// TIA Portal V16 export
// export: Created 2022-11-17T15:49:43.8022431Z, ExportSetting WithDefaults, DisplayName Totally Integrated Automation Portal, DisplayVersion V16 Update 6, DisplayName TIA Portal Version Control Interface, DisplayVersion V16 Update 2, DisplayName TIA Portal Openness, DisplayVersion V16 Update 6, DisplayName SINAMICS Startdrive Advanced, DisplayVersion V16 Update 5, DisplayName SINAMICS Startdrive G130, G150, S120, S150, SINAMICS MV, S210, DisplayVersion V16 Update 5, DisplayName SINAMICS Startdrive G110M, G120, G120C, G120D, G120P, G115D, DisplayVersion V16 Update 5, DisplayName STEP 7 Professional, DisplayVersion V16 Update 6, DisplayName STEP 7 Safety, DisplayVersion V16, DisplayName WinCC Advanced, DisplayVersion V16 Update 6
DATA_BLOCK "DB237_Program13"   // DB237
{ S7_Optimized_Access := 'FALSE' }
AUTHOR : Robopac
VERSION : 0.0
// stored: AutoNumber false, IsOnlyStoredInLoadMemory false, IsWriteProtectedInAS false
   VAR RETAIN
      Program13 { S7_SetPoint := 'True'} : "DatiProgramma";
   END_VAR
BEGIN
   Program13.Wrapping := TRUE;
   Program13.TopLenght := 500;
   Program13.TopRelease := 0;
   Program13.TopDown := 0;
   Program13.Top := 4;
   Program13.PressurePTime := 0;
   Program13.LifterTime := 0;
   Program13.RevOverContrast := 1;
   Program13.RopeEndCycle := 16#02;
   Program13.Spare4 := 16#01;
   Program13.RopeTime := 1500;
   Program13.RevOverClamp := 1;
   Program13.FilmForceFinalRev := 10;
   Program13.FilmPrestretchFinalRev := 100;
   Program13.ArmSpeed := 100;
   Program13.CarriageDown4Top := 500;
   Program13.TopDownTime := 1500;
   Program13.LapsUnderTop := 0;
   Program13.Spare6 := 0;
   Program13.Spare7 := 0;
   Program13.Spare8 := 0;
   Program13.Spare9 := 0;
   Program13.Spare10 := 0;
   Program13.Spare11 := 0;
   Program13.Spare12 := 0;
   Program13.Overlap0_1 := 0;
   Program13.Height1 := 130;
   Program13.Landmark1 := FALSE;
   Program13.Lifter1 := FALSE;
   Program13.SpareBit1H1 := FALSE;
   Program13.Airblower1 := TRUE;
   Program13.NextStep1 := TRUE;
   Program13.PressureP1 := TRUE;
   Program13.SpareByte2H1 := 16#00;
   Program13.Revolution1 := 1;
   Program13.RopeUnit1_1 := 16#01;
   Program13.RopeUnit1_2 := 16#01;
   Program13.FilmForce1 := 5;
   Program13.FilmPrestretch1 := 200;
   Program13.Spare3H1 := 0;
   Program13.Spare49 := 0;
   Program13.Spare50 := 0;
   Program13.Spare51 := 0;
   Program13.Spare52 := 0;
   Program13.Spare53 := 0;
   Program13.Overlap1_2 := 0;
   Program13.Height2 := 50;
   Program13.Landmark2 := FALSE;
   Program13.Lifter2 := FALSE;
   Program13.SpareBit1H2 := FALSE;
   Program13.Airblower2 := TRUE;
   Program13.NextStep2 := TRUE;
   Program13.PressureP2 := TRUE;
   Program13.SpareByte2H2 := 16#00;
   Program13.Revolution2 := 1;
   Program13.RopeUnit2_1 := 16#01;
   Program13.RopeUnit2_2 := 16#01;
   Program13.FilmForce2 := 20;
   Program13.FilmPrestretch2 := 200;
   Program13.Spare3H2 := 0;
   Program13.Spare54 := 0;
   Program13.Spare55 := 0;
   Program13.Spare56 := 0;
   Program13.Spare57 := 0;
   Program13.Spare58 := 0;
   Program13.Overlap2_3 := 100;
   Program13.Height3 := -50;
   Program13.Landmark3 := TRUE;
   Program13.Lifter3 := FALSE;
   Program13.SpareBit1H3 := FALSE;
   Program13.Airblower3 := TRUE;
   Program13.NextStep3 := TRUE;
   Program13.PressureP3 := TRUE;
   Program13.SpareByte2H3 := 16#00;
   Program13.Revolution3 := 2;
   Program13.RopeUnit3_1 := 16#01;
   Program13.RopeUnit3_2 := 16#01;
   Program13.FilmForce3 := 30;
   Program13.FilmPrestretch3 := 200;
   Program13.Spare3H3 := 0;
   Program13.Spare59 := 0;
   Program13.Spare60 := 0;
   Program13.Spare61 := 380;
   Program13.Spare62 := 2800;
   Program13.Spare63 := 0;
   Program13.Overlap3_4 := 100;
   Program13.Height4 := 100;
   Program13.Landmark4 := FALSE;
   Program13.Lifter4 := FALSE;
   Program13.SpareBit1H4 := FALSE;
   Program13.Airblower4 := TRUE;
   Program13.NextStep4 := TRUE;
   Program13.PressureP4 := TRUE;
   Program13.SpareByte2H4 := 16#00;
   Program13.Revolution4 := 3;
   Program13.RopeUnit4_1 := 16#02;
   Program13.RopeUnit4_2 := 16#02;
   Program13.FilmForce4 := 30;
   Program13.FilmPrestretch4 := 200;
   Program13.Spare3H4 := 0;
   Program13.Spare64 := 0;
   Program13.Spare65 := 0;
   Program13.Spare66 := 0;
   Program13.Spare67 := 0;
   Program13.Spare68 := 0;
   Program13.Overlap4_5 := 0;
   Program13.Height5 := 50;
   Program13.Landmark5 := FALSE;
   Program13.Lifter5 := FALSE;
   Program13.SpareBit1H5 := FALSE;
   Program13.Airblower5 := TRUE;
   Program13.NextStep5 := FALSE;
   Program13.PressureP5 := FALSE;
   Program13.SpareByte2H5 := 16#00;
   Program13.Revolution5 := 1;
   Program13.RopeUnit5_1 := 16#01;
   Program13.RopeUnit5_2 := 16#01;
   Program13.FilmForce5 := 30;
   Program13.FilmPrestretch5 := 200;
   Program13.Spare3H5 := 0;
   Program13.Spare69 := 0;
   Program13.Spare70 := 0;
   Program13.Spare71 := 0;
   Program13.Spare72 := 0;
   Program13.Spare73 := 0;
   Program13.Overlap5_6 := 100;
   Program13.Height6 := 50;
   Program13.Landmark6 := FALSE;
   Program13.Lifter6 := FALSE;
   Program13.SpareBit1H6 := FALSE;
   Program13.Airblower6 := TRUE;
   Program13.NextStep6 := FALSE;
   Program13.PressureP6 := FALSE;
   Program13.SpareByte2H6 := 16#00;
   Program13.Revolution6 := 2;
   Program13.RopeUnit6_1 := 16#02;
   Program13.RopeUnit6_2 := 16#01;
   Program13.FilmForce6 := 20;
   Program13.FilmPrestretch6 := 200;
   Program13.Spare3H6 := 0;
   Program13.Spare74 := 0;
   Program13.Spare75 := 0;
   Program13.Spare76 := 0;
   Program13.Spare77 := 0;
   Program13.Spare78 := 0;
   Program13.Overlap6_7 := 0;
   Program13.Height7 := 0;
   Program13.Landmark7 := FALSE;
   Program13.Lifter7 := FALSE;
   Program13.SpareBit1H7 := FALSE;
   Program13.Airblower7 := FALSE;
   Program13.NextStep7 := TRUE;
   Program13.PressureP7 := FALSE;
   Program13.SpareByte2H7 := 16#00;
   Program13.Revolution7 := 1;
   Program13.RopeUnit7_1 := 16#01;
   Program13.RopeUnit7_2 := 16#01;
   Program13.FilmForce7 := 0;
   Program13.FilmPrestretch7 := 100;
   Program13.Spare3H7 := 0;
   Program13.Spare79 := 0;
   Program13.Spare80 := 0;
   Program13.Spare81 := 0;
   Program13.Spare82 := 0;
   Program13.Spare83 := 0;
   Program13.Overlap7_8 := 0;
   Program13.Height8 := 0;
   Program13.Landmark8 := FALSE;
   Program13.Lifter8 := FALSE;
   Program13.SpareBit1H8 := FALSE;
   Program13.Airblower8 := FALSE;
   Program13.NextStep8 := TRUE;
   Program13.PressureP8 := FALSE;
   Program13.SpareByte2H8 := 16#00;
   Program13.Revolution8 := 1;
   Program13.RopeUnit8_1 := 16#01;
   Program13.RopeUnit8_2 := 16#01;
   Program13.FilmForce8 := 0;
   Program13.FilmPrestretch8 := 100;
   Program13.Spare3H8 := 0;
   Program13.Spare84 := 0;
   Program13.Spare85 := 0;
   Program13.Spare86 := 0;
   Program13.Spare87 := 0;
   Program13.Spare88 := 0;
   Program13.Overlap8_9 := 0;
   Program13.Height9 := 0;
   Program13.Landmark9 := FALSE;
   Program13.Lifter9 := FALSE;
   Program13.SpareBit1H9 := FALSE;
   Program13.Airblower9 := FALSE;
   Program13.NextStep9 := TRUE;
   Program13.PressureP9 := FALSE;
   Program13.SpareByte2H9 := 16#00;
   Program13.Revolution9 := 1;
   Program13.RopeUnit9_1 := 16#01;
   Program13.RopeUnit9_2 := 16#01;
   Program13.FilmForce9 := 0;
   Program13.FilmPrestretch9 := 100;
   Program13.Spare3H9 := 0;
   Program13.Spare89 := 0;
   Program13.Spare90 := 0;
   Program13.Spare91 := 0;
   Program13.Spare92 := 0;
   Program13.Spare93 := 0;
   Program13.Overlap9_10 := 0;
   Program13.Height10 := 0;
   Program13.Landmark10 := FALSE;
   Program13.Lifter10 := FALSE;
   Program13.SpareBit1H10 := FALSE;
   Program13.Airblower10 := FALSE;
   Program13.NextStep10 := FALSE;
   Program13.PressureP10 := FALSE;
   Program13.SpareByte2H10 := 16#00;
   Program13.Revolution10 := 1;
   Program13.RopeUnit10_1 := 16#01;
   Program13.RopeUnit10_2 := 16#01;
   Program13.FilmForce10 := 0;
   Program13.FilmPrestretch10 := 100;
   Program13.Spare3H10 := 0;
   Program13.Spare94 := 0;
   Program13.Spare95 := 0;
   Program13.Spare96 := 0;
   Program13.Spare97 := 0;
   Program13.Spare98 := 0;
   Program13.Overlap10_11 := 0;
   Program13.Height11 := 0;
   Program13.Landmark11 := FALSE;
   Program13.Lifter11 := FALSE;
   Program13.SpareBit1H11 := FALSE;
   Program13.Airblower11 := FALSE;
   Program13.NextStep11 := TRUE;
   Program13.PressureP11 := FALSE;
   Program13.SpareByte2H11 := 16#00;
   Program13.Revolution11 := 1;
   Program13.RopeUnit11_1 := 16#01;
   Program13.RopeUnit11_2 := 16#01;
   Program13.FilmForce11 := 0;
   Program13.FilmPrestretch11 := 100;
   Program13.Spare3H11 := 0;
   Program13.Spare99 := 0;
   Program13.Spare100 := 0;
   Program13.Spare101 := 0;
   Program13.Spare102 := 0;
   Program13.Spare103 := 0;
   Program13.Overlap11_12 := 0;
   Program13.Height12 := 0;
   Program13.Landmark12 := FALSE;
   Program13.Lifter12 := FALSE;
   Program13.SpareBit1H12 := FALSE;
   Program13.Airblower12 := FALSE;
   Program13.NextStep12 := FALSE;
   Program13.PressureP12 := FALSE;
   Program13.SpareByte2H12 := 16#00;
   Program13.Revolution12 := 1;
   Program13.RopeUnit12_1 := 16#01;
   Program13.RopeUnit12_2 := 16#01;
   Program13.FilmForce12 := 0;
   Program13.FilmPrestretch12 := 100;
   Program13.Spare3H12 := 0;
   Program13.Spare104 := 0;
   Program13.Spare105 := 0;
   Program13.Spare106 := 0;
   Program13.Spare107 := 0;
   Program13.Spare108 := 0;
END_DATA_BLOCK
